{attribute 'qualified_only'}
VAR_GLOBAL
	/// Inputs
	stInputs	:	stIOinput;
	/// Outputs
	stOutputs	: 	stIOoutput;
	
	bHomeSwitch: BOOL;
END_VAR

(* stored: Version 1.1.0.1, ProductVersion 3.1.4024.12
   GVL gvlIO: Id {ec8b3721-9de7-4a16-b80d-24d091a4ea63} *)
